FUNCTION_BLOCK FB_ScannerImplementation
VAR
	_Keyence : BOOL;
	_scannerCognex : BOOL;
END_VAR

_Keyence:= TRUE;

END_FUNCTION_BLOCK

(* stored: Version 1.1.0.1, ProductVersion 3.1.4024.12
   POU FB_ScannerImplementation: Id {bbe3db64-5932-4d33-8d44-3c0350c6f67c}, SpecialFunc None *)
